FUNCTION_BLOCK FB_FindDestination
VAR_IN_OUT
	RoundRobin		:	ST_RoundRobin;
	aDiverts		:	ARRAY[*] OF ST_Divert;
	DestinationID	:	DINT;
END_VAR
VAR_INPUT
	SorterLogEnable	:	UDINT;
END_VAR
VAR_OUTPUT
	DestinationIndex	:	DINT;
	DestinationState	:	DINT;
END_VAR
VAR
	DivertArrayMin		:	DINT;
	DivertArrayMax		:	DINT;
	Last_Enabled	:	UINT;
	IndexCheck		:	DINT;
	sMessage		:	STRING;
END_VAR

// Get the upper and lower bounds of the divert array
DivertArrayMin := LOWER_BOUND(aDiverts,1);
DivertArrayMax := UPPER_BOUND(aDiverts,1);

//When a response is received, find the designated Destination
IF DestinationID >= 0 THEN
	IF SorterLogEnable.SORTER_DESTINATION_LU THEN
		sMessage := CONCAT(' Destination: ', DINT_TO_STRING(DestinationID));
		// Write to the Error List
		ADSLOGSTR( msgCtrlMask := ADSLOG_MSGTYPE_HINT OR ADSLOG_MSGTYPE_LOG
			, msgFmtStr := 'Lookup: %s'
			, strArg := sMessage);
	END_IF
	// Check to see if the Destination is defined as a round-robin destination for this sorter
	IF DestinationID = RoundRobin.Destination THEN
		// Test to see if the last enabled round robin destinations are still enabled
		// If they are different, restart the round-robin assignment to accommodate differences 
		IF RoundRobin.Enabled = Last_Enabled THEN
			// Test to see if the round robin assignments have all been met
			// If they have, clear and start over
			IF RoundRobin.Available = RoundRobin.Sent THEN
				RoundRobin.Sent := 0;
			END_IF
		ELSE
			// Capture the new enabled round-robin destinations
			// Restart the round robin assignments
			Last_Enabled := RoundRobin.Enabled;
			RoundRobin.Sent := 0;
		END_IF
		FOR IndexCheck := 0 TO 15 DO
			IF (
			   ((RoundRobin.Enabled AND LREAL_TO_UINT(EXPT(2,IndexCheck))) > 0) 
			   AND ((RoundRobin.Available AND LREAL_TO_UINT(EXPT(2,IndexCheck))) > 0)
			   AND NOT ((RoundRobin.Sent AND LREAL_TO_UINT(EXPT(2,IndexCheck))) > 0))
			   THEN
				RoundRobin.Sent := LREAL_TO_UINT(EXPT(2,IndexCheck)) OR RoundRobin.Sent;
				IF RoundRobin.aDestinations[IndexCheck] >= DivertArrayMin
				   AND RoundRobin.aDestinations[IndexCheck] <= DivertArrayMax
				   THEN
					DestinationIndex := RoundRobin.aDestinations[IndexCheck];
					DestinationID := aDiverts[DestinationIndex].Config.Number;
				ELSE
					DestinationIndex := DivertArrayMax;
				END_IF
				DestinationState := 0;
				EXIT;
			END_IF
		END_FOR
		IF SorterLogEnable.SORTER_DESTINATION_LU THEN
			sMessage := DINT_TO_STRING(DestinationIndex);
			sMessage := CONCAT(' Dest ID: ', DINT_TO_STRING(DestinationID));
			// Write to the Error List
			ADSLOGSTR( msgCtrlMask := ADSLOG_MSGTYPE_HINT OR ADSLOG_MSGTYPE_LOG
				, msgFmtStr := 'RoundRobin Dest: %s'
				, strArg := sMessage);
		END_IF
	ELSE
		DestinationIndex := DivertArrayMax;
		FOR IndexCheck := DivertArrayMin TO DivertArrayMax  DO
			IF aDiverts[IndexCheck].Config.Number = DestinationID THEN
				DestinationIndex := IndexCheck;
				DestinationState := 0;
				EXIT;
			END_IF
		END_FOR
		IF SorterLogEnable.SORTER_DESTINATION_LU THEN
			sMessage := DINT_TO_STRING(DestinationIndex);
			sMessage := CONCAT(' Dest ID: ', DINT_TO_STRING(DestinationID));
			// Write to the Error List
			ADSLOGSTR( msgCtrlMask := ADSLOG_MSGTYPE_HINT OR ADSLOG_MSGTYPE_LOG
				, msgFmtStr := 'Lookup Dest: %s'
				, strArg := sMessage);
		END_IF
	END_IF
END_IF

END_FUNCTION_BLOCK

(* stored: Version 1.1.0.1, ProductVersion 3.1.4024.4
   POU FB_FindDestination: Id {56bb7952-67df-4bb2-8615-b0884b2a1363}, SpecialFunc None *)
